RoboDK station: Gui.20x20square.rdk

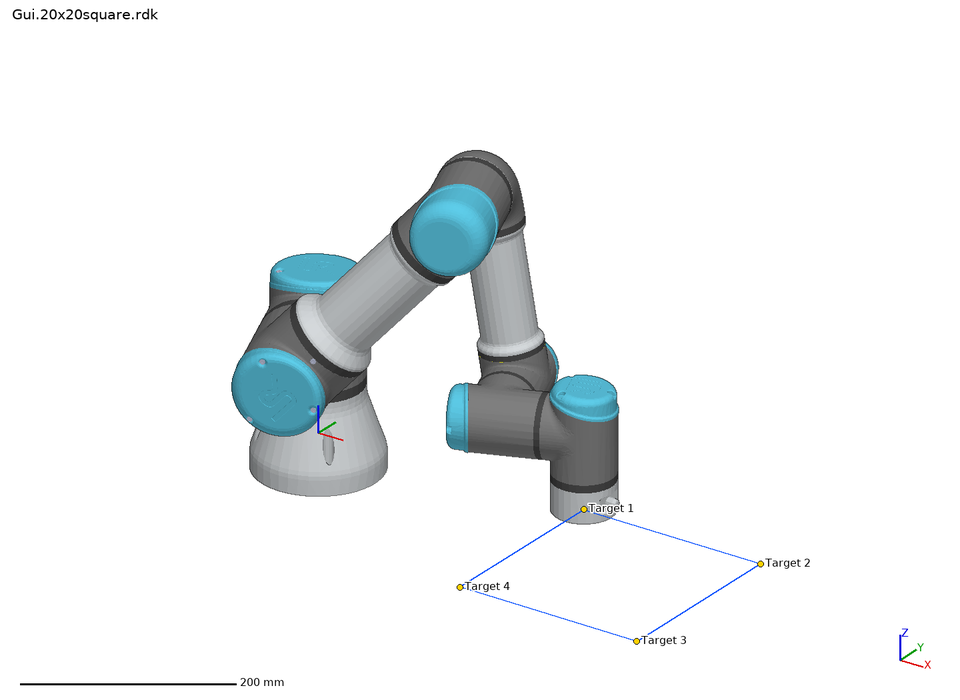
[picture v0: the station drawn from its stored meshes, robots at their saved joint values, targets as dots, program paths as lines]
Station Gui. Poses are relative to the parent item; angles as X-Y-Z fixed-axis rotations.
  - frame UR3 Base at (0, 0, 0) mm
    - robot UR3: 6 axes, payload 3 kg, reach 500 mm, repeatability 0.1 mm, weight 11 kg
        modified DH rows (alpha deg, a mm, theta deg, d mm): 0, 0, 0, 118; 90, 0, 180, 0; 0, 243.65, 0, 0; 0, 213, 0, 110.4; -90, 0, 0, 83.4; 90, 0, 180, 82.4
        joint limits [-360, -360, -360, -360, -360, -360] to [360, 360, 360, 360, 360, 360]; home [0, -90, -90, 0, 90, 0]; saved at [21.597, -132.336, -129.161, -8.535, 89.986, 21.597]
    - target Target 1 (Cartesian target) at (300, 0, 5) mm, rotated rx 179.97 ry -0.03 rz -90 deg; joints [21.597, -132.336, -129.161, -8.535, 89.986, 21.597] of UR3
    - target Target 2 (Cartesian target) at (500, 0, 5) mm, rotated rx 179.97 ry -0.03 rz -90 deg; joints [12.759, -158.861, -54.918, -56.251, 89.981, 12.759] of UR3
    - target Target 3 (Cartesian target) at (500, -200, 5) mm, rotated rx 179.97 ry -0.03 rz -90 deg; joints [-9.967, -171.7, -26.277, -72.043, 89.971, -9.967] of UR3
    - target Target 4 (Cartesian target) at (300, -200, 5) mm, rotated rx 179.97 ry -0.03 rz -90 deg; joints [-15.853, -137.004, -110.458, -22.556, 89.969, -15.853] of UR3
    - target Target 5 (Cartesian target) at (300, 0, 5) mm, rotated rx 179.97 ry -0.03 rz -90 deg; joints [21.597, -132.336, -129.161, -8.535, 89.986, 21.597] of UR3
  - program Prog1 (6 instructions, listed below)
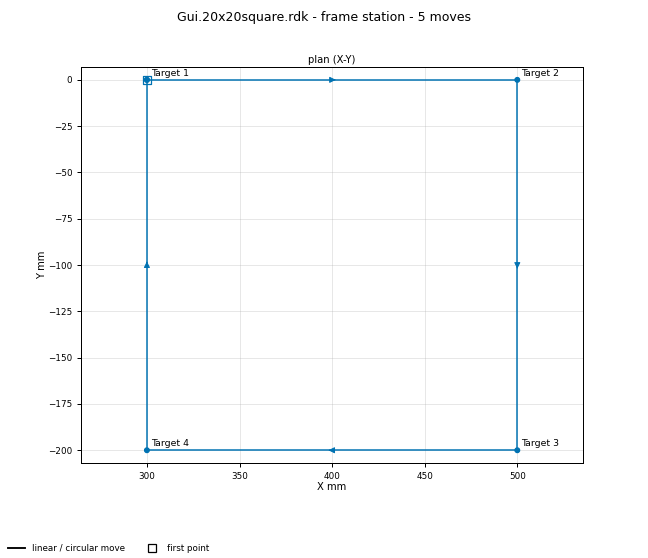
[picture p0: tool path of Gui.20x20square.rdk in frame station, 5 of 5 moves have a stored position in this frame; points joined in program order, loops and branches not executed]

--- program Prog1 (robot UR3) ---
  Referenz erstellen.: UR3 Base
  MoveL (Target 1)
  MoveL (Target 2)
  MoveL (Target 3)
  MoveL (Target 4)
  MoveL (Target 5)
